{attribute 'qualified_only'}
VAR_GLOBAL
    // TRUE = 數位孿生模擬模式；使用時在 DAS_CoreSys 傳入 MachineControl(EnableSimulation := GVL_SimMode.bSimMode)
    bSimMode : BOOL := FALSE;
END_VAR

(* stored: Version 1.1.0.1, ProductVersion 3.1.4024.13
   GVL GVL_SimMode: Id {a1b2c3d4-e5f6-7890-abcd-ef1234567890} *)
